FUNCTION_BLOCK ASR_SWITCH (* Switching (demultiplexing) ASR events (SET/RESET) based on boolean input G *)
  (* Standard: 61499-1 Annex A; Description: Copyright (c) 2017 fortiss GmbH This program and the accompanying materials are made available under the terms of the Eclipse Public License 2.0 which is available at https://www.eclipse.org/legal/epl-2.0/ SPDX-License-Identifier: EPL-2.0 *)
  (* Version 3.0, 2025-04-14, Patrick Aigner, changed package *)
  (* Version 1.0, 2017-09-21, Alois Zoitl, fortiss GmbH, initial API and implementation and/or initial documentation *)
  PACKAGE adapter::events::unidirectional;
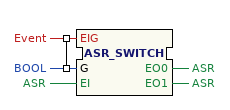
  EVENT_INPUT
    EIG WITH G; (* set G *)
  END_EVENT
  VAR_INPUT
    G : BOOL; (* Switch EI to EO0 when G=0, to EO1 when G=1 *)
  END_VAR
  SOCKETS
    EI : adapter::types::unidirectional::ASR; (* Event Input *)
  END_SOCKETS
  PLUGS
    EO0 : adapter::types::unidirectional::ASR; (* Output, switched from EI when G=0 *)
    EO1 : adapter::types::unidirectional::ASR; (* Output, switched from EI when G=1 *)
  END_PLUGS
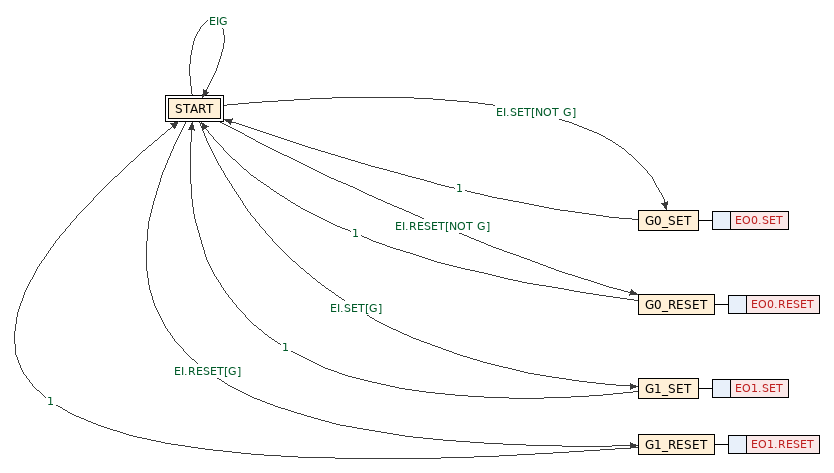
  EC_STATES
    START; (* Initial State *)
    G0_SET : -> EO0.SET; (* Issue EO0 when EI arrives with G=0 *)
    G1_SET : -> EO1.SET; (* Issue EO1 when EI arrives with G=1 *)
    G0_RESET : -> EO0.RESET;
    G1_RESET : -> EO1.RESET;
  END_STATES
  EC_TRANSITIONS
    G0_SET TO START := 1;
    START TO G0_SET := EI.SET[NOT G];
    START TO G1_SET := EI.SET[G];
    START TO START := EIG;
    START TO G0_RESET := EI.RESET[NOT G];
    G0_RESET TO START := 1;
    START TO G1_RESET := EI.RESET[G];
    G1_SET TO START := 1;
    G1_RESET TO START := 1;
  END_TRANSITIONS
END_FUNCTION_BLOCK
